// TIA Portal project "TestIOSL" (V18)

(* hardware
DEVICE "S7-1500/ET200MP station_1"  S7-1500 station
   slot 0: "Rail_0"  Rack  6ES7 590-1***0-0AA0
   slot 1: "PLC_1"  CPU 1516F-3 PN/DP  6ES7 516-3FN01-0AB0  V2.9
      slot 3: "CPU display_1"  6ES7591-1BA00-0AA0
      slot 32768: "PROFINET interface_1"  X1
      slot 33024: "PROFINET interface_2"  X2
      slot 33280: "DP interface_1"  X3
      slot 34817: "Virtual CP interface port_1"  Virtual CP interface port  Virtual CP interface port
DEVICE "GSD device_1"  GSD.Device.PN
   slot 0: "Rack"  Rack  V1.0
   slot 0: "IOL_IO32_PQI"  IOL_IO32_PQI
   slot 0: "pdp67pn"  PDP67 PN 8FDIO 4IOLS V1.0.x  4R000004  V1.0.x
      slot 0: "PDP67 PN 8FDIO 4IOLS V1.0.x"  PDP67 PN 8FDIO 4IOLS V1.0.x
      slot 1: "PROFINET IO"  PROFINET IO
         slot 1: "X21"  X21
         slot 2: "X22"  X22
      slot 1: "Port 2FDIO_1"  Port 2FDIO
         slot 0: "Port 2FDIO"  Port 2FDIO
      slot 2: "Port 2FDIO_2"  Port 2FDIO
         slot 0: "Port 2FDIO"  Port 2FDIO
      slot 3: "Port 2FDIO_3"  Port 2FDIO
         slot 0: "Port 2FDIO"  Port 2FDIO
      slot 4: "Port 2FDIO_4"  Port 2FDIO
         slot 0: "Port 2FDIO"  Port 2FDIO
      slot 11: "Container FS FDIO channel-granular_1"  Container FS FDIO channel-granular
         slot 0: "Container FS FDIO channel-granular"  Container FS FDIO channel-granular
   slot 1: "IOLS_SP3"  IOLS_SP3
   slot 5: "Port IOL_1"  Port IOL
*)

// ===== PLC "PLC_1"  CPU 1516F-3 PN/DP =====

VAR_GLOBAL   // PLC tag table "Default tag table"
   "mPDP67SafetyReset" AT %M100.1 : Bool;
   "PITgateboxButton1Status" AT %I0.7 : Bool;
   "PITgateboxButton2Status" AT %I2.7 : Bool;
   "PITgateboxButton3Status" AT %I4.7 : Bool;
   "PITgateboxButton1LEDFlash" AT %Q3.7 : Bool;
   "PITgateboxButton2LEDFlash" AT %Q5.7 : Bool;
   "PITgateboxButton3LEDFlash" AT %Q7.7 : Bool;
   "PITgateboxButton1LEDON" AT %Q9.7 : Bool;
   "PITgateboxButton2LEDON" AT %Q11.7 : Bool;
   "PITgateboxButton3LEDON" AT %Q13.7 : Bool;
   "PITgateboxSetLockingTrigger" AT %Q0.0 : Bool;
   "PITgateboxSetLockingDevice" AT %Q2.0 : Bool;
   "PITgateboxSafetyRelease1" AT %I100.0 : Bool;   // 1=Safety Outpout ON,1
   "PITgateboxSafetyRelease2" AT %I100.1 : Bool;   // 1=Safety Outpout ON,2
   "PITgateboxSafetyESTOP" AT %I100.2 : Bool;
   "PITgateboxSafetyPowerOutput32" AT %Q100.0 : Bool;
   "PITgateboxSafetyPowerOutput42" AT %Q100.1 : Bool;
   "PITgateboxLockInPosition" AT %I9.0 : Bool;   // 1=Door Lock Position OK
   "PITgateboxLockStatus1" AT %I11.0 : Bool;   // 1=Safety Output is OK
END_VAR

DATA_BLOCK "Main_Safety_RTG1_DB"   // DB1, F_DB
{ S7_Optimized_Access := 'TRUE' }
NAME : FUSI
VERSION : 0.1
// stored: InstanceOfName Main_Safety_RTG1
"Main_Safety_RTG1"
BEGIN
END_DATA_BLOCK

FUNCTION_BLOCK "Main_Safety_RTG1"   // FB1, F_FBD
{ S7_Optimized_Access := 'TRUE' }
   VAR
      SFDOOR_Instance : SFDOOR;
      P_TRIG_Bit1 : Bool;
      iDoorStep : Int;
      DoorLock : Bool;
      OutputIsOK : Bool;
      TriggerLock : Bool;
      TriggerLocked : Bool;
      ResetTrigger : Bool;
      DoorUnlock : Bool;
      TON1 : TON;
      TON2 : TON;
   END_VAR
   VAR_TEMP
      DoorLockInPosition : Bool;
   END_VAR
BEGIN

REGION Network 1: QBAD and Reset for IOLink Safety, Channel1,1=Acknowledgment for reintegration
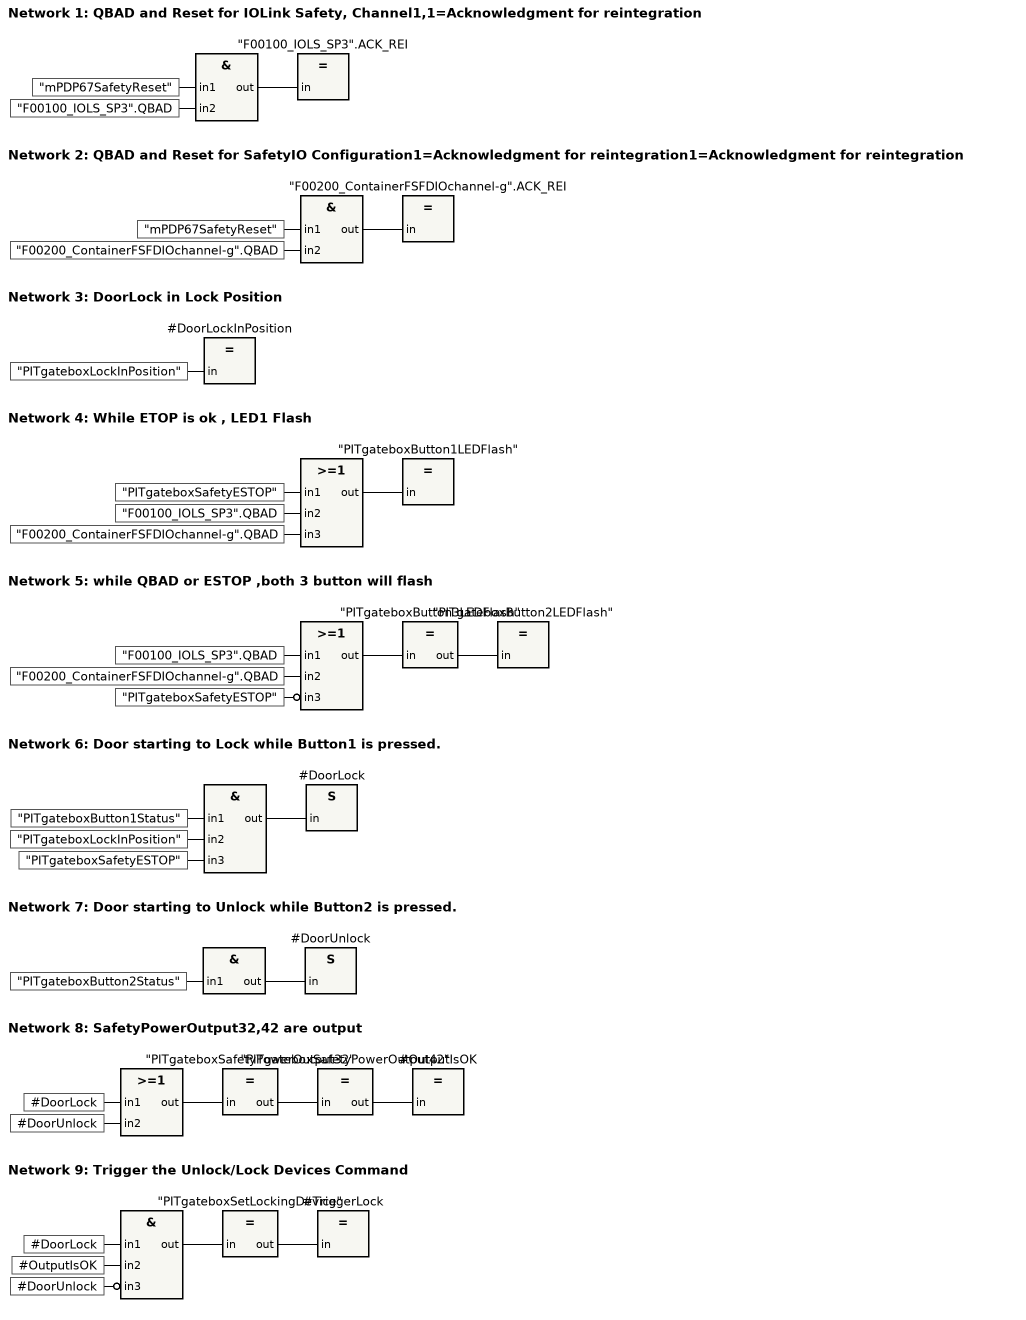
   "F00100_IOLS_SP3".ACK_REI := "mPDP67SafetyReset" AND "F00100_IOLS_SP3".QBAD;
END_REGION

REGION Network 2: QBAD and Reset for SafetyIO Configuration1=Acknowledgment for reintegration1=Acknowledgment for reintegration
   "F00200_ContainerFSFDIOchannel-g".ACK_REI := "mPDP67SafetyReset" AND "F00200_ContainerFSFDIOchannel-g".QBAD;
END_REGION

REGION Network 3: DoorLock in Lock Position
   #DoorLockInPosition := "PITgateboxLockInPosition";
END_REGION

REGION Network 4: While ETOP is ok , LED1 Flash
   "PITgateboxButton1LEDFlash" := "PITgateboxSafetyESTOP" OR "F00100_IOLS_SP3".QBAD OR "F00200_ContainerFSFDIOchannel-g".QBAD;
END_REGION

REGION Network 5: while QBAD or ESTOP ,both 3 button will flash
   "PITgateboxButton3LEDFlash" := "F00100_IOLS_SP3".QBAD OR "F00200_ContainerFSFDIOchannel-g".QBAD OR NOT "PITgateboxSafetyESTOP";
   "PITgateboxButton2LEDFlash" := "PITgateboxButton3LEDFlash";
END_REGION

REGION Network 6: Door starting to Lock while Button1 is pressed.
   IF "PITgateboxButton1Status" AND "PITgateboxLockInPosition" AND "PITgateboxSafetyESTOP" THEN
       #DoorLock := TRUE;
   END_IF;
END_REGION

REGION Network 7: Door starting to Unlock while Button2 is pressed.
   IF "PITgateboxButton2Status" THEN #DoorUnlock := TRUE; END_IF;
END_REGION

REGION Network 8: SafetyPowerOutput32,42 are output
   "PITgateboxSafetyPowerOutput32" := #DoorLock OR #DoorUnlock;
   "PITgateboxSafetyPowerOutput42" := "PITgateboxSafetyPowerOutput32";
   #OutputIsOK := "PITgateboxSafetyPowerOutput32";
END_REGION

REGION Network 9: Trigger the Unlock/Lock Devices Command
   "PITgateboxSetLockingDevice" := #DoorLock AND #OutputIsOK AND NOT #DoorUnlock;
   #TriggerLock := "PITgateboxSetLockingDevice";
END_REGION

REGION Network 10: Trigger the Unlock/Lock Command
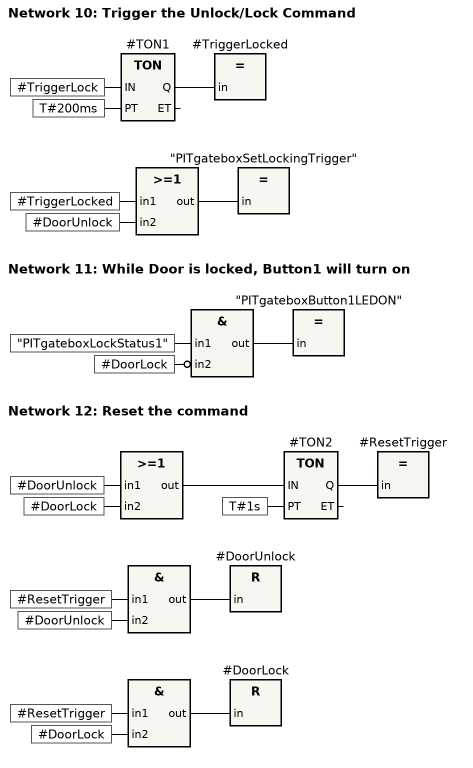
   #TON1.TON(IN := #TriggerLock, PT := T#200ms);
   #TriggerLocked := #TON1.Q;
   "PITgateboxSetLockingTrigger" := #TriggerLocked OR #DoorUnlock;
END_REGION

REGION Network 11: While Door is locked, Button1 will turn on
   "PITgateboxButton1LEDON" := "PITgateboxLockStatus1" AND NOT #DoorLock;
END_REGION

REGION Network 12: Reset the command
   #TON2.TON(IN := #DoorUnlock OR #DoorLock, PT := T#1s);
   #ResetTrigger := #TON2.Q;
   IF #ResetTrigger AND #DoorUnlock THEN #DoorUnlock := FALSE; END_IF;
   IF #ResetTrigger AND #DoorLock THEN #DoorLock := FALSE; END_IF;
END_REGION
END_FUNCTION_BLOCK

ORGANIZATION_BLOCK "Main"   // OB1, LAD, ProgramCycle
TITLE = "Main Program Sweep (Cycle)"
{ S7_Optimized_Access := 'TRUE' }
VERSION : 0.1
   VAR_INPUT
      Initial_Call : Bool;   // Initial call of this OB
      Remanence : Bool;   // =True, if remanent data are available
   END_VAR
BEGIN
END_ORGANIZATION_BLOCK